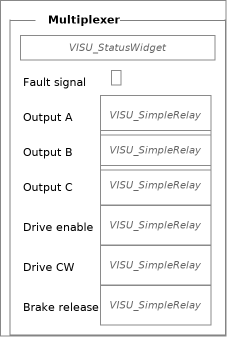
VISUALIZATION VISU_M2Multiplexer  // 227x337
VAR_IN_OUT
	ref : M2Multiplexer;
    widget : M2MultiplexerWidget;
END_VAR
    Polyline (120,20) (225,20) (225,335) (10,335) (10,20) (35,20)
    Frame (100,95 111x40)
        shows VISU_SimpleRelay(ref := ref.parts.A, widget := widget.A)
    Label (20,105 75x25), "Output A"
    Label (20,140 75x25), "Output B"
    Frame (100,130 111x40)
        shows VISU_SimpleRelay(ref := ref.parts.B, widget := widget.B)
    Label (20,175 75x25), "Output C"
    Frame (100,165 111x40)
        shows VISU_SimpleRelay(ref := ref.parts.C, widget := widget.C)
    Label (20,215 85x25), "Drive enable"
    Frame (100,205 111x40)
        shows VISU_SimpleRelay(ref := ref.parts.driveEnable, widget := widget.driveEnable)
    Label (20,255 85x25), "Drive CW"
    Frame (100,245 111x40)
        shows VISU_SimpleRelay(ref := ref.parts.CW, widget := widget.CW)
    Label (20,295 95x25), "Brake release"
    Frame (100,285 111x40)
        shows VISU_SimpleRelay(ref := ref.parts.release, widget := widget.release)
    Frame (111,70 10x15)
        shows VISU_State_red_green(state := ref.noFault)
    Label (20,70 75x25), "Fault signal"
    Frame (20,35 195x25)
        shows VISU_StatusWidget(widget := widget.actualStatus)
    Label (45,10 150x20), "Multiplexer"
END_VISUALIZATION

(* stored: Version 1.1.0.1, ProductVersion 3.1.4019.2
   Visu VISU_M2Multiplexer: Id {0a3e715f-5f96-4da7-8f27-89350390f163} *)
